{attribute 'linkalways'}
{attribute 'no_explicit_call' := 'This FB is a CLASS and must be accessed using methods or properties'}
{attribute 'enable_dynamic_creation'}
FUNCTION_BLOCK _GVCP_REGISTER_VALUE EXTENDS AliasDatatypeBase
VAR
	localData : GVCP_REGISTER_VALUE;
	activeData : REFERENCE TO GVCP_REGISTER_VALUE REF= localData;
	aliasBaseDatatype : _UDINT(0);
END_VAR

PROPERTY PUBLIC Address : PVOID
GET
Address := ADR(activeData);
END_GET
END_PROPERTY

METHOD PUBLIC ClearReference
VAR_INPUT
END_VAR
activeData REF= localData;
SetBaseDatatypeReference();
END_METHOD

METHOD PUBLIC Clone : I_Datatype
VAR
    pClone : POINTER TO _GVCP_REGISTER_VALUE;
END_VAR
pClone := __NEW(_GVCP_REGISTER_VALUE(InitialValue := Value));
IF pClone = 0 THEN
    RETURN;
END_IF
pClone^.TryCopyFrom(THIS^);
Clone := pClone^;
END_METHOD

METHOD FB_init : BOOL
VAR_INPUT
	bInitRetains : BOOL; // if TRUE, the retain variables are initialized (warm start / cold start)
	bInCopyCode : BOOL;  // if TRUE, the instance afterwards gets moved into the copy code (online change)
	InitialValue : GVCP_REGISTER_VALUE := 0;
END_VAR
localData := InitialValue;
SetBaseDatatypeReference();
AddBaseDatatype(aliasBaseDatatype);
END_METHOD

PROPERTY PUBLIC Identifier : T_MAXSTRING
GET
Identifier := 'GVCP_REGISTER_VALUE';
END_GET
END_PROPERTY

METHOD PUBLIC MakeReferenceTo
VAR_INPUT
	ReferenceTarget : REFERENCE TO GVCP_REGISTER_VALUE;
END_VAR
activeData REF= ReferenceTarget;
SetBaseDatatypeReference();
END_METHOD

METHOD PROTECTED SetBaseDatatypeReference
VAR_INPUT
END_VAR
aliasBaseDatatype.MakeReferenceTo(activeData);
END_METHOD

PROPERTY PUBLIC Size : UDINT
GET
Size := SIZEOF(activeData);
END_GET
END_PROPERTY

METHOD TryMakeReferenceTo : BOOL
VAR_INPUT
	Target : I_Datatype;
END_VAR
VAR
	pTargetData : POINTER TO GVCP_REGISTER_VALUE;
END_VAR
IF NOT IsEquivalentTo(Target) THEN
	RETURN;
END_IF

pTargetData := Target.Address;
activeData REF= pTargetData^;
SetBaseDatatypeReference();
TryMakeReferenceTo := TRUE;
END_METHOD

PROPERTY PUBLIC Value : REFERENCE TO GVCP_REGISTER_VALUE
GET
Value REF= activeData;
END_GET
END_PROPERTY

END_FUNCTION_BLOCK

(* stored: Version 1.1.0.1, ProductVersion 3.1.4026.19
   POU _GVCP_REGISTER_VALUE: Id {bab2ea4d-620d-4f6f-81f7-52bab10d0f7d}, SpecialFunc None
   Folder Core: Id {689359eb-0e74-4af4-a396-80e1e1edd64a}
   Folder Protected: Id {e016778e-24fa-425b-82ca-7ee9970794c8}
   Folder Customize: Id {eeb174ab-305a-4afc-8ec3-f2399ba82a11}
   Folder Constructor: Id {8593887b-a43a-48a5-94fd-92ef266706c6}
   Property Address: Id {dfa2c8ab-ecd9-43cd-b7bc-d662f5cd02ea}
   Get Get: Id {3d563e18-128d-464c-8902-09f64a25be94}
   Method ClearReference: Id {5c5480b7-0079-4f51-88c5-e34e164d84fd}
   Method Clone: Id {f68ba939-7d38-4958-9946-92b4edc723b5}
   Method FB_init: Id {f5deea25-c21c-4884-94e5-5ca00bc0544b}
   Property Identifier: Id {db906bdd-7364-4a88-8a5c-57fc526866bc}
   Get Get: Id {a5e8bb45-b956-413e-96d4-8450608cacb8}
   Method MakeReferenceTo: Id {97219a8e-8b13-4ce8-858f-8300340aea3b}
   Method SetBaseDatatypeReference: Id {69e2ea0d-ce59-4f95-8c09-10fe75a04aaf}
   Property Size: Id {a5ebf132-0288-4f27-8da9-9a97c2d7855f}
   Get Get: Id {f9a27caf-acf6-4dde-bf34-9c0cd3403105}
   Method TryMakeReferenceTo: Id {9da506e2-9255-4878-9206-baa5ababff5f}
   Property Value: Id {f1ab5142-2216-4a96-9fc7-5715ae5a0572}
   Get Get: Id {eaf0d061-4f39-45c6-b7cd-343141bef64c} *)
